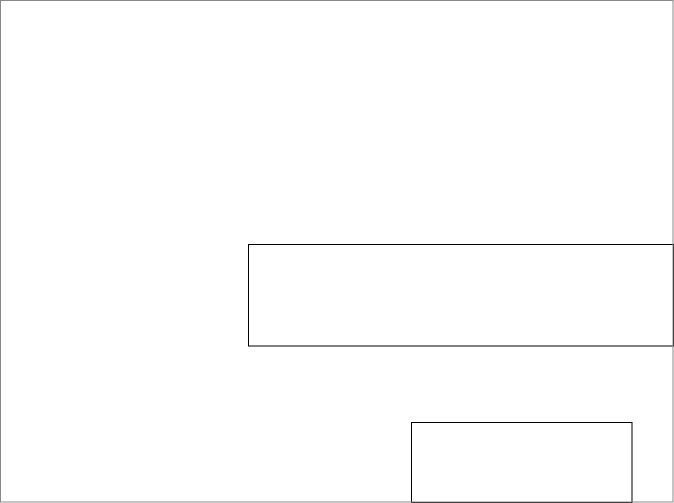
VISUALIZATION Visualization  // 674x503
    Rectangle (248,244 426x102)
    Rectangle (411,422 221x81)
        OnMouseClick: ChangeLanguage ChangeLanguage=CATALÀ
END_VISUALIZATION

(* stored: Version 1.1.0.1
   Visu Visualization: Id {3d191336-253b-4049-9c07-50d572e30d01} *)
